ABB RobotStudio station: Montaje_Herramienta.rsstnx

Station Montaje_Herramienta (saved by RobotStudio 23.4.10609.1)
Controller Controlador1
  mechanical unit ROB_1: IRB140_6_81_C_03, 6 joints, base frame (0, 0, 0) mm
Layout (positions relative to the parent item):
  - IRB140_6_81_C_03 [mechanism, from %ABB.RobotStudio.Models.IRB140%\IRB140_6_81_C_G_03.rslib] at (0, 0, 0) mm; joint values [0, 0.0169, -0.0078, 0, 0.5145, 0] (rad or m)
  - FinalTool [mechanism] at (512.35, 0, 676) mm, rotated rx 180 ry 60 rz 180 deg
      TCP FinalTool at (175, 27.22, 27.22) mm, rotated rx -90 ry 45 rz -90 deg
      links: Support_RS
  - Logo_names [part] at (1000, -125, 230) mm, rotated rx 0 ry 0 rz 180 deg, size 357.3 x 250 x 190.4 mm
Attachment: FinalTool is attached to IRB140_6_81_C_03 / Link6
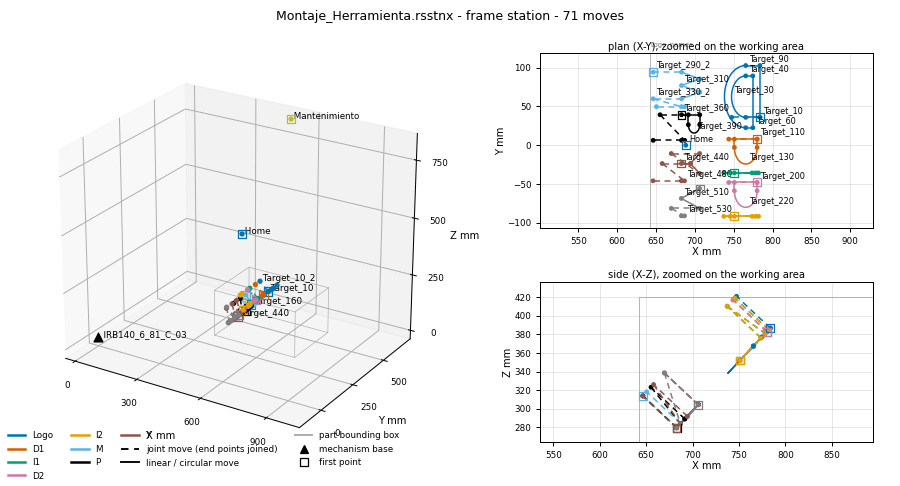
[picture p0: tool path of Montaje_Herramienta.rsstnx in frame station, 71 of 71 moves have a stored position in this frame; points joined in program order, loops and branches not executed]
Targets, tools, work objects and paths stored in the station, written as RAPID:
! task T_ROB1
MODULE Module1
  CONST robtarget Home:=[[688.354427157,0,618.841978046],[0.5,0,0.866025404,0],[0,0,0,0],[9E+09,9E+09,9E+09,9E+09,9E+09,9E+09]];
  PERS tooldata FinalTool:=[TRUE,[[-38.5,0,181],[1,0,0,0]],[1,[0,0,1],[1,0,0,0],0,0,0]];
  TASK PERS wobjdata Workobject_1:=[FALSE,TRUE,"",[[822.628,-125,413.586],[0.396843374,0,0.917886342,0]],[[0,0,-10],[1,0,0,0]]];
  CONST robtarget Mantenimiento:=[[491.434141762,691.445179965,824.691178836],[0.866840807,-0.149108085,0.220825114,0.42141436],[0,-1,0,1],[9E+09,9E+09,9E+09,9E+09,9E+09,9E+09]];
  CONST robtarget Target_10:=[[46.091,160.915,0],[1,0,0,0],[0,-1,0,0],[9E+09,9E+09,9E+09,9E+09,9E+09,9E+09]];
  CONST robtarget Target_20:=[[72.767,160.915,0],[1,0,0,0],[0,0,0,0],[9E+09,9E+09,9E+09,9E+09,9E+09,9E+09]];
  CONST robtarget Target_30:=[[99.443,187.591,0],[1,0,0,0],[0,-1,0,0],[9E+09,9E+09,9E+09,9E+09,9E+09,9E+09]];
  CONST robtarget Target_40:=[[72.767,214.267,0],[1,0,0,0],[0,-1,0,0],[9E+09,9E+09,9E+09,9E+09,9E+09,9E+09]];
  CONST robtarget Target_50:=[[59.429,214.267,0],[1,0,0,0],[0,-1,0,0],[9E+09,9E+09,9E+09,9E+09,9E+09,9E+09]];
  CONST robtarget Target_60:=[[59.429,147.577,0],[1,0,0,0],[0,-1,0,0],[9E+09,9E+09,9E+09,9E+09,9E+09,9E+09]];
  CONST robtarget Target_70:=[[72.767,147.577,0],[1,0,0,0],[0,-1,0,0],[9E+09,9E+09,9E+09,9E+09,9E+09,9E+09]];
  CONST robtarget Target_80:=[[112.781,187.591,0],[1,0,0,0],[0,-1,0,0],[9E+09,9E+09,9E+09,9E+09,9E+09,9E+09]];
  CONST robtarget Target_90:=[[72.767,227.605,0],[1,0,0,0],[0,-1,0,0],[9E+09,9E+09,9E+09,9E+09,9E+09,9E+09]];
  CONST robtarget Target_100:=[[46.091,227.605,0],[1,0,0,0],[0,-1,0,0],[9E+09,9E+09,9E+09,9E+09,9E+09,9E+09]];
  CONST robtarget Target_110:=[[51.426,132.866,0],[1,0,0,0],[0,0,0,0],[9E+09,9E+09,9E+09,9E+09,9E+09,9E+09]];
  CONST robtarget Target_120:=[[51.426,122.195,0],[1,0,0,0],[-1,0,-1,0],[9E+09,9E+09,9E+09,9E+09,9E+09,9E+09]];
  CONST robtarget Target_130:=[[72.767,100.855,0],[1,0,0,0],[-1,0,-1,0],[9E+09,9E+09,9E+09,9E+09,9E+09,9E+09]];
  CONST robtarget Target_140:=[[94.108,122.195,0],[1,0,0,0],[-1,0,-1,0],[9E+09,9E+09,9E+09,9E+09,9E+09,9E+09]];
  CONST robtarget Target_150:=[[94.108,132.866,0],[1,0,0,0],[0,-1,0,0],[9E+09,9E+09,9E+09,9E+09,9E+09,9E+09]];
  CONST robtarget Target_160:=[[94.108,89.421,0],[1,0,0,0],[0,0,0,0],[9E+09,9E+09,9E+09,9E+09,9E+09,9E+09]];
  CONST robtarget Target_170:=[[60.763,89.421,0],[1,0,0,0],[-1,0,-1,0],[9E+09,9E+09,9E+09,9E+09,9E+09,9E+09]];
  CONST robtarget Target_180:=[[54.094,89.421,0],[1,0,0,0],[-1,0,-1,0],[9E+09,9E+09,9E+09,9E+09,9E+09,9E+09]];
  CONST robtarget Target_190:=[[48.759,89.421,0],[1,0,0,0],[-1,0,-1,0],[9E+09,9E+09,9E+09,9E+09,9E+09,9E+09]];
  CONST robtarget Target_200:=[[51.426,77.138,0],[1,0,0,0],[0,0,0,0],[9E+09,9E+09,9E+09,9E+09,9E+09,9E+09]];
  CONST robtarget Target_210:=[[51.426,66.467,0],[1,0,0,0],[-1,0,-1,0],[9E+09,9E+09,9E+09,9E+09,9E+09,9E+09]];
  CONST robtarget Target_220:=[[72.767,45.127,0],[1,0,0,0],[-1,0,-1,0],[9E+09,9E+09,9E+09,9E+09,9E+09,9E+09]];
  CONST robtarget Target_230:=[[94.108,66.467,0],[1,0,0,0],[-1,0,-1,0],[9E+09,9E+09,9E+09,9E+09,9E+09,9E+09]];
  CONST robtarget Target_240:=[[94.108,77.138,0],[1,0,0,0],[-1,0,-1,0],[9E+09,9E+09,9E+09,9E+09,9E+09,9E+09]];
  CONST robtarget Target_250:=[[94.108,33.511,0],[1,0,0,0],[0,0,0,0],[9E+09,9E+09,9E+09,9E+09,9E+09,9E+09]];
  CONST robtarget Target_260:=[[60.763,33.511,0],[1,0,0,0],[-1,0,-1,0],[9E+09,9E+09,9E+09,9E+09,9E+09,9E+09]];
  CONST robtarget Target_270:=[[54.094,33.511,0],[1,0,0,0],[-1,0,-1,0],[9E+09,9E+09,9E+09,9E+09,9E+09,9E+09]];
  CONST robtarget Target_280:=[[48.759,33.511,0],[1,0,0,0],[-1,0,-1,0],[9E+09,9E+09,9E+09,9E+09,9E+09,9E+09]];
  CONST robtarget Target_290:=[[193.374,219.018,0],[1,0,0,0],[0,0,0,0],[9E+09,9E+09,9E+09,9E+09,9E+09,9E+09]];
  CONST robtarget Target_300:=[[159.174,210.468,0],[1,0,0,0],[0,-1,1,0],[9E+09,9E+09,9E+09,9E+09,9E+09,9E+09]];
  CONST robtarget Target_310:=[[193.374,201.918,0],[1,0,0,0],[0,-2,1,0],[9E+09,9E+09,9E+09,9E+09,9E+09,9E+09]];
  CONST robtarget Target_320:=[[159.174,193.368,0],[1,0,0,0],[0,-1,1,0],[9E+09,9E+09,9E+09,9E+09,9E+09,9E+09]];
  CONST robtarget Target_330:=[[193.374,184.818,0],[1,0,0,0],[0,-2,1,0],[9E+09,9E+09,9E+09,9E+09,9E+09,9E+09]];
  CONST robtarget Target_340:=[[193.374,174.678,0],[1,0,0,0],[0,-2,1,0],[9E+09,9E+09,9E+09,9E+09,9E+09,9E+09]];
  CONST robtarget Target_350:=[[187.389,174.678,0],[1,0,0,0],[0,-2,1,0],[9E+09,9E+09,9E+09,9E+09,9E+09,9E+09]];
  CONST robtarget Target_360:=[[193.374,164.249,0],[1,0,0,0],[0,-2,1,0],[9E+09,9E+09,9E+09,9E+09,9E+09,9E+09]];
  CONST robtarget Target_370:=[[159.174,164.249,0],[1,0,0,0],[0,-2,1,0],[9E+09,9E+09,9E+09,9E+09,9E+09,9E+09]];
  CONST robtarget Target_380:=[[159.174,151.424,0],[1,0,0,0],[0,-2,1,0],[9E+09,9E+09,9E+09,9E+09,9E+09,9E+09]];
  CONST robtarget Target_390:=[[169.861,140.736,0],[1,0,0,0],[0,-2,1,0],[9E+09,9E+09,9E+09,9E+09,9E+09,9E+09]];
  CONST robtarget Target_400:=[[180.549,151.424,0],[1,0,0,0],[0,-2,1,0],[9E+09,9E+09,9E+09,9E+09,9E+09,9E+09]];
  CONST robtarget Target_410:=[[180.549,164.249,0],[1,0,0,0],[0,-2,1,0],[9E+09,9E+09,9E+09,9E+09,9E+09,9E+09]];
  CONST robtarget Target_420:=[[187.389,131.33,0],[1,0,0,0],[0,-2,1,0],[9E+09,9E+09,9E+09,9E+09,9E+09,9E+09]];
  CONST robtarget Target_430:=[[193.374,131.33,0],[1,0,0,0],[0,-2,1,0],[9E+09,9E+09,9E+09,9E+09,9E+09,9E+09]];
  CONST robtarget Target_440:=[[193.651,101.513,0],[1,0,0,0],[-1,1,-2,0],[9E+09,9E+09,9E+09,9E+09,9E+09,9E+09]];
  CONST robtarget Target_450:=[[176.551,101.513,0],[1,0,0,0],[-1,1,-2,0],[9E+09,9E+09,9E+09,9E+09,9E+09,9E+09]];
  CONST robtarget Target_460:=[[159.451,114.338,0],[1,0,0,0],[-1,1,-2,0],[9E+09,9E+09,9E+09,9E+09,9E+09,9E+09]];
  CONST robtarget Target_470:=[[159.451,88.688,0],[1,0,0,0],[-1,1,-2,0],[9E+09,9E+09,9E+09,9E+09,9E+09,9E+09]];
  CONST robtarget Target_480:=[[187.666,79.24,0],[1,0,0,0],[-1,1,-2,0],[9E+09,9E+09,9E+09,9E+09,9E+09,9E+09]];
  CONST robtarget Target_490:=[[193.651,79.24,0],[1,0,0,0],[-1,1,-2,0],[9E+09,9E+09,9E+09,9E+09,9E+09,9E+09]];
  CONST robtarget Target_500:=[[159.451,69.411,0],[1,0,0,0],[-1,1,-2,0],[9E+09,9E+09,9E+09,9E+09,9E+09,9E+09]];
  CONST robtarget Target_510:=[[193.651,56.586,0],[1,0,0,0],[-1,1,-2,0],[9E+09,9E+09,9E+09,9E+09,9E+09,9E+09]];
  CONST robtarget Target_520:=[[159.451,43.761,0],[1,0,0,0],[-1,0,-2,0],[9E+09,9E+09,9E+09,9E+09,9E+09,9E+09]];
  CONST robtarget Target_530:=[[187.666,34.148,0],[1,0,0,0],[-1,1,-2,0],[9E+09,9E+09,9E+09,9E+09,9E+09,9E+09]];
  CONST robtarget Target_540:=[[193.651,34.148,0],[1,0,0,0],[-1,1,-2,0],[9E+09,9E+09,9E+09,9E+09,9E+09,9E+09]];
  CONST robtarget Target_10_2:=[[46.091,160.915,-50],[1,0,0,0],[0,-1,0,0],[9E+09,9E+09,9E+09,9E+09,9E+09,9E+09]];
  CONST robtarget Target_110_2:=[[51.426,132.866,-50],[1,0,0,0],[0,-1,0,0],[9E+09,9E+09,9E+09,9E+09,9E+09,9E+09]];
  CONST robtarget Target_170_2:=[[60.763,89.421,-50],[1,0,0,0],[-1,0,-1,0],[9E+09,9E+09,9E+09,9E+09,9E+09,9E+09]];
  CONST robtarget Target_190_2:=[[48.759,89.421,-50],[1,0,0,0],[-1,0,-1,0],[9E+09,9E+09,9E+09,9E+09,9E+09,9E+09]];
  CONST robtarget Target_200_2:=[[51.426,77.138,-50],[1,0,0,0],[-1,0,-1,0],[9E+09,9E+09,9E+09,9E+09,9E+09,9E+09]];
  CONST robtarget Target_260_2:=[[60.763,33.511,-50],[1,0,0,0],[-1,0,-1,0],[9E+09,9E+09,9E+09,9E+09,9E+09,9E+09]];
  CONST robtarget Target_280_2:=[[48.759,33.511,-50],[1,0,0,0],[-1,0,-1,0],[9E+09,9E+09,9E+09,9E+09,9E+09,9E+09]];
  CONST robtarget Target_290_2:=[[193.374,219.018,-50],[1,0,0,0],[0,-1,1,0],[9E+09,9E+09,9E+09,9E+09,9E+09,9E+09]];
  CONST robtarget Target_330_2:=[[193.374,184.818,-50],[1,0,0,0],[0,-1,0,0],[9E+09,9E+09,9E+09,9E+09,9E+09,9E+09]];
  CONST robtarget Target_350_2:=[[187.389,174.678,-50],[1,0,0,0],[0,-1,0,0],[9E+09,9E+09,9E+09,9E+09,9E+09,9E+09]];
  CONST robtarget Target_410_2:=[[180.549,164.249,-50],[1,0,0,0],[0,-1,0,0],[9E+09,9E+09,9E+09,9E+09,9E+09,9E+09]];
  CONST robtarget Target_460_2:=[[159.451,114.338,-50],[1,0,0,0],[-1,0,-1,0],[9E+09,9E+09,9E+09,9E+09,9E+09,9E+09]];
  CONST robtarget Target_450_2:=[[176.551,101.513,-50],[1,0,0,0],[-1,0,-1,0],[9E+09,9E+09,9E+09,9E+09,9E+09,9E+09]];
  CONST robtarget Target_490_2:=[[193.651,79.24,-50],[1,0,0,0],[-1,0,-1,0],[9E+09,9E+09,9E+09,9E+09,9E+09,9E+09]];
  CONST robtarget Target_520_2:=[[159.451,43.761,-50],[1,0,0,0],[-1,0,-1,0],[9E+09,9E+09,9E+09,9E+09,9E+09,9E+09]];
  CONST robtarget Target_430_2:=[[193.374,131.33,-50],[1,0,0,0],[0,-1,0,0],[9E+09,9E+09,9E+09,9E+09,9E+09,9E+09]];
  PROC Logo()
    MoveJ Target_10,v100,fine,FinalTool\WObj:=Workobject_1;
    MoveL Target_20,v100,fine,FinalTool\WObj:=Workobject_1;
    MoveC Target_30,Target_40,v100,fine,FinalTool\WObj:=Workobject_1;
    MoveL Target_50,v100,fine,FinalTool\WObj:=Workobject_1;
    MoveL Target_60,v100,fine,FinalTool\WObj:=Workobject_1;
    MoveL Target_70,v100,fine,FinalTool\WObj:=Workobject_1;
    MoveC Target_80,Target_90,v100,fine,FinalTool\WObj:=Workobject_1;
    MoveL Target_100,v100,fine,FinalTool\WObj:=Workobject_1;
    MoveL Target_10,v100,fine,FinalTool\WObj:=Workobject_1;
    MoveJ Target_10_2,v200,z10,FinalTool\WObj:=Workobject_1;
  ENDPROC
  PROC D1()
    MoveJ Target_110,v100,fine,FinalTool\WObj:=Workobject_1;
    MoveL Target_120,v100,fine,FinalTool\WObj:=Workobject_1;
    MoveC Target_130,Target_140,v100,fine,FinalTool\WObj:=Workobject_1;
    MoveL Target_150,v100,fine,FinalTool\WObj:=Workobject_1;
    MoveL Target_110,v100,fine,FinalTool\WObj:=Workobject_1;
    MoveJ Target_110_2,v200,z10,FinalTool\WObj:=Workobject_1;
  ENDPROC
  PROC I1()
    MoveJ Target_160,v100,fine,FinalTool\WObj:=Workobject_1;
    MoveL Target_170,v100,fine,FinalTool\WObj:=Workobject_1;
    MoveJ Target_170_2,v200,z10,FinalTool\WObj:=Workobject_1;
    MoveJ Target_180,v100,fine,FinalTool\WObj:=Workobject_1;
    MoveL Target_190,v100,fine,FinalTool\WObj:=Workobject_1;
    MoveJ Target_190_2,v200,z10,FinalTool\WObj:=Workobject_1;
  ENDPROC
  PROC D2()
    MoveJ Target_200,v100,fine,FinalTool\WObj:=Workobject_1;
    MoveL Target_210,v100,fine,FinalTool\WObj:=Workobject_1;
    MoveC Target_220,Target_230,v100,fine,FinalTool\WObj:=Workobject_1;
    MoveL Target_240,v100,fine,FinalTool\WObj:=Workobject_1;
    MoveL Target_200,v100,fine,FinalTool\WObj:=Workobject_1;
    MoveJ Target_200_2,v200,z10,FinalTool\WObj:=Workobject_1;
  ENDPROC
  PROC I2()
    MoveJ Target_250,v100,fine,FinalTool\WObj:=Workobject_1;
    MoveL Target_260,v100,fine,FinalTool\WObj:=Workobject_1;
    MoveJ Target_260_2,v200,z10,FinalTool\WObj:=Workobject_1;
    MoveJ Target_270,v100,fine,FinalTool\WObj:=Workobject_1;
    MoveL Target_280,v100,fine,FinalTool\WObj:=Workobject_1;
    MoveJ Target_280_2,v200,z10,FinalTool\WObj:=Workobject_1;
  ENDPROC
  PROC M()
    MoveJ Target_290_2,v200,z10,FinalTool\WObj:=Workobject_1;
    MoveJ Target_290,v100,fine,FinalTool\WObj:=Workobject_1;
    MoveL Target_300,v100,fine,FinalTool\WObj:=Workobject_1;
    MoveL Target_310,v100,fine,FinalTool\WObj:=Workobject_1;
    MoveL Target_320,v100,fine,FinalTool\WObj:=Workobject_1;
    MoveL Target_330,v100,fine,FinalTool\WObj:=Workobject_1;
    MoveJ Target_330_2,v200,z10,FinalTool\WObj:=Workobject_1;
    MoveJ Target_340,v100,fine,FinalTool\WObj:=Workobject_1;
    MoveL Target_350,v100,fine,FinalTool\WObj:=Workobject_1;
    MoveJ Target_350_2,v200,z10,FinalTool\WObj:=Workobject_1;
  ENDPROC
  PROC P()
    MoveJ Target_360,v100,fine,FinalTool\WObj:=Workobject_1;
    MoveL Target_370,v100,fine,FinalTool\WObj:=Workobject_1;
    MoveL Target_380,v100,fine,FinalTool\WObj:=Workobject_1;
    MoveC Target_390,Target_400,v100,fine,FinalTool\WObj:=Workobject_1;
    MoveL Target_410,v100,fine,FinalTool\WObj:=Workobject_1;
    MoveJ Target_410_2,v200,z10,FinalTool\WObj:=Workobject_1;
    MoveJ Target_420,v100,fine,FinalTool\WObj:=Workobject_1;
    MoveJ Target_430,v100,fine,FinalTool\WObj:=Workobject_1;
    MoveJ Target_430_2,v200,z10,FinalTool\WObj:=Workobject_1;
  ENDPROC
  PROC Y()
    MoveJ Target_440,v100,fine,FinalTool\WObj:=Workobject_1;
    MoveL Target_450,v100,fine,FinalTool\WObj:=Workobject_1;
    MoveL Target_460,v100,fine,FinalTool\WObj:=Workobject_1;
    MoveJ Target_460_2,v200,z10,FinalTool\WObj:=Workobject_1;
    MoveJ Target_470,v100,fine,FinalTool\WObj:=Workobject_1;
    MoveL Target_450,v100,fine,FinalTool\WObj:=Workobject_1;
    MoveJ Target_450_2,v200,z10,FinalTool\WObj:=Workobject_1;
    MoveJ Target_480,v100,fine,FinalTool\WObj:=Workobject_1;
    MoveL Target_490,v100,fine,FinalTool\WObj:=Workobject_1;
    MoveJ Target_490_2,v200,z10,FinalTool\WObj:=Workobject_1;
  ENDPROC
  PROC V()
    MoveJ Target_500,v100,fine,FinalTool\WObj:=Workobject_1;
    MoveL Target_510,v100,fine,FinalTool\WObj:=Workobject_1;
    MoveL Target_520,v100,fine,FinalTool\WObj:=Workobject_1;
    MoveJ Target_520_2,v200,z10,FinalTool\WObj:=Workobject_1;
    MoveJ Target_530,v100,fine,FinalTool\WObj:=Workobject_1;
    MoveL Target_540,v100,fine,FinalTool\WObj:=Workobject_1;
  ENDPROC
  PROC Main()
    GoEscritura;
    GoMantenimeinto;
    Homing;
  ENDPROC
  PROC GoMantenimeinto()
    Homing;
    SetDO DO_03,0;
    SetDO DO_02,1;
    MoveJ Mantenimiento,v200,z10,FinalTool\WObj:=wobj0;
  ENDPROC
  PROC GoEscritura()
    Homing;
    SetDO DO_03,0;
    SetDO DO_01,1;
    Logo;
    D1;
    I1;
    D2;
    I2;
    M;
    P;
    Y;
    V;
  ENDPROC
  PROC Homing()
    SetDO DO_01,0;
    SetDO DO_02,0;
    SetDO DO_03,1;
    MoveJ Home,v300,z10,FinalTool\WObj:=wobj0;
  ENDPROC
ENDMODULE

